FUNCTION_BLOCK FB_Divide
VAR_INPUT
	nDivIn1:		INT;
	nDivIn2:		INT;
END_VAR
VAR_OUTPUT
	nDivOut:		INT;
END_VAR
VAR
END_VAR

nDivOut:= nDivIn1 / nDivIn2;

END_FUNCTION_BLOCK

(* stored: Version 1.1.0.1, ProductVersion 3.1.4024.3
   POU FB_Divide: Id {046f7d88-e44d-4d9d-8555-4308ed1dbdef}, SpecialFunc None *)
